FUNCTION ToAnyType : __SYSTEM.AnyType
VAR_INPUT
	object		: ANY;
END_VAR

ToAnyType := object;

END_FUNCTION

(* stored: Version 1.1.0.1, ProductVersion 3.1.4024.15
   POU ToAnyType: Id {443949fb-0e92-45a1-919c-47897b524390}, SpecialFunc None *)
